(* PLC project Traffic control simulator, CODESYS CODESYS V3.5 SP14 Patch 1, author Toni Kucic *)
(* stored: creationDateTime 2019-08-10T15:27:01.2415123, version 1.0, modificationDateTime 2019-08-10T15:27:01.0436346, organization TK Automation *)

FUNCTION_BLOCK CollisionDetection
  VAR_INPUT
    xcor1 : REAL := 0;  (* X Coordinate of object 1 *)
    ycor1 : REAL := 0;  (* Y Coordinate of object 1 *)
    height1 : REAL := 0;  (* Height of object 1 *)
    width1 : REAL := 0;  (* Width of object 1 *)
    xcor2 : REAL := 0;  (* X Coordinate of object 2 *)
    ycor2 : REAL := 0;  (* Y Coordinate of object 2 *)
    height2 : REAL := 0;  (* Height of object 1 *)
    width2 : REAL := 0;  (* Width of object 1 *)
  END_VAR
  VAR_OUTPUT
    isCollision : BOOL := FALSE;
  END_VAR

            IF xcor1 < (xcor2 + width2) AND
   (xcor1 + width1) > xcor2 AND
   ycor1 < (ycor2 + height2) AND
  ( height1 + ycor1) > ycor2 THEN
   isCollision := TRUE;
ELSE
	isCollision := FALSE;
END_IF
          
END_FUNCTION_BLOCK

FUNCTION_BLOCK MoveSprite
  VAR_IN_OUT
    xCor : INT := 0;
    yCor : INT := 0;
  END_VAR
  VAR_INPUT
    xScreen : INT := 0;  (* Width of the screen *)
    yScreen : INT := 0;  (* Height of the screen *)
    SpriteWidth : INT := 0;  (* Width of the sprite *)
    SpriteHeight : INT := 0;  (* Height of the sprite *)
    ySpeed : INT := 0;  (* Control up or down movement with +- *)
    xSpeed : INT := 0;  (* Control left or right movement with +- *)
  END_VAR

            (* Reseting the position if sprite goes off screen *)
(* If moving left to right *)
IF xCor >= xScreen  AND xSpeed > 0 THEN
	xCor := -SpriteWidth;
(* If moving right to left *)
ELSIF xCor <= -SpriteWidth AND xSpeed < 0 THEN
	xCor := xScreen;	
END_IF
(* If moving from up, down *)
IF yCor >= yScreen AND ySpeed > 0 THEN
	yCor := -SpriteHeight;
(* If moving from down, up *)
ELSIF yCor < -SpriteHeight AND ySpeed < 0 THEN
	yCor := yScreen;	
END_IF

(* Actual moving of the coordinates *)
xCor := xCor + xSpeed;
yCor := yCor + ySpeed;

          
END_FUNCTION_BLOCK

PROGRAM xc03_TrafficControl
  VAR
    vSequenceA : DINT := 1;
    TimerA : TOF;
    vSequenceB : DINT := 0;
    TimerB : TOF;
    Start : BOOL;
    StartOld : BOOL;
    vSequence : DINT := 0;
    TactTimer : TON;
    vPeriodTime : TIME := TIME#1m25s0ms;
    vElapsedTime : TIME;
  END_VAR

                    
TactTimer(IN:=TRUE, PT:=vPeriodTime, ET => vElapsedTime);
IF TactTimer.Q THEN
	TactTimer(IN:=FALSE);
END_IF
(* Direction Up, Down traffic light *)
xgv03.TLight3Red := vElapsedTime <= T#5S OR vElapsedTime >= T#37S AND vElapsedTime <= T#85S;
xgv03.TLight3Yellow := vElapsedTime > T#3S AND vElapsedTime <= T#5S OR vElapsedTime >= T#35S AND vElapsedTime <= T#37S;
xgv03.TLight3Green := vElapsedTime >= T#5S AND vElapsedTime <= T#35S;

(* Mirror the other side of the Up, Down direction *)
xgv03.TLight4Red := xgv03.TLight3Red;
xgv03.TLight4Yellow := xgv03.TLight3Yellow;
xgv03.TLight4Green := xgv03.TLight3Green;

(* Direction Left, Right traffic light *)
xgv03.TLight2Red := vElapsedTime >= T#0S AND vElapsedTime <= T#39S OR vElapsedTime >= T#71S AND vElapsedTime <= T#85S;
xgv03.TLight2Yellow := vElapsedTime > T#37S AND vElapsedTime <= T#39S OR vElapsedTime >= T#69S AND vElapsedTime <= T#71S;
xgv03.TLight2Green := vElapsedTime >= T#39S AND vElapsedTime <= T#69S;

(* Mirror the other side of the Left, Right direction *)
xgv03.TLight1Red := xgv03.TLight2Red;
xgv03.TLight1Yellow := xgv03.TLight2Yellow;
xgv03.TLight1Green := xgv03.TLight2Green;
(*CASE vSequence OF
	0:
	(* Starting sequence, direction Up, Down *)
	TimerA
	Task03GVL.TLight1Red := TRUE;
	
END_CASE
CASE vSequenceA OF
	0: TimerA(IN:=FALSE,PT:=T#20S);
	Task03GVL.TLight1Yellow:= FALSE;
	Task03GVL.TLight1Red:= FALSE;
	Task03GVL.TLight1Green:= TimerA.Q;
	Task03GVL.TLight2Green := Task03GVL.TLight1Green;
	IF NOT TimerA.Q THEN
		TimerA(IN:=TRUE);
		vSequenceA:=1;
	END_IF
	1: TimerA(IN:=FALSE,PT:=T#4S);
	Task03GVL.TLight1Red:= FALSE;
	Task03GVL.TLight1Green:= FALSE;
	Task03GVL.TLight1Yellow:= TimerA.Q;
	Task03GVL.TLight2Yellow := Task03GVL.TLight1Yellow;
	IF NOT TimerA.Q THEN
		TimerA(IN:=TRUE);
		vSequenceA:=2;
	END_IF
		2: TimerA(IN:=FALSE,PT:=T#30S);
	Task03GVL.TLight1Green:= FALSE;
	Task03GVL.TLight1Yellow:= FALSE;
	Task03GVL.TLight1Red:= TimerA.Q;
	Task03GVL.TLight2Red := Task03GVL.TLight1Red;
	IF NOT TimerA.Q THEN
		TimerA(IN:=TRUE);
		vSequenceA:=3;
	END_IF
		3: TimerA(IN:=FALSE,PT:=T#4S);
	Task03GVL.TLight1Green:= FALSE;
	Task03GVL.TLight1Red:= TimerA.Q;
	Task03GVL.TLight1Yellow:= TimerA.Q;
	Task03GVL.TLight2Red := Task03GVL.TLight1Red;
	Task03GVL.TLight2Yellow := Task03GVL.TLight1Yellow;
	IF NOT TimerA.Q THEN
		TimerA(IN:=TRUE);
		vSequenceA:=0;
		IF vSequenceB=6 THEN
		vSequenceB:=3;	
		END_IF
		
	END_IF
END_CASE

CASE vSequenceB OF
	0: TimerB(IN:=FALSE,PT:=T#4S);
	Task03GVL.TLight3Green:= FALSE;
	Task03GVL.TLight3Red:= TimerB.Q;
	Task03GVL.TLight3Yellow:= TimerB.Q;
	Task03GVL.TLight4Red := Task03GVL.TLight3Red;
	Task03GVL.TLight4Yellow := Task03GVL.TLight3Yellow;
	IF NOT TimerB.Q THEN
		TimerB(IN:=TRUE);
		vSequenceB:=1;
	END_IF
	
	1: TimerB(IN:=FALSE,PT:=T#20S);
	Task03GVL.TLight3Yellow:= FALSE;
	Task03GVL.TLight3Red:= FALSE;
	Task03GVL.TLight3Green:= TimerB.Q;
	Task03GVL.TLight4Green := Task03GVL.TLight3Green;
	IF NOT TimerB.Q THEN
		TimerB(IN:=TRUE);
		vSequenceB:=2;
	END_IF
	
	2: TimerB(IN:=FALSE,PT:=T#4S);
	Task03GVL.TLight3Red:= FALSE;
	Task03GVL.TLight3Green:= FALSE;
	Task03GVL.TLight3Yellow:= TimerB.Q;
	Task03GVL.TLight4Yellow := Task03GVL.TLight3Yellow;
	IF NOT TimerB.Q THEN
		TimerB(IN:=TRUE);
		vSequenceB:=3;
	END_IF
	
		3: TimerB(IN:=FALSE,PT:=T#30S);
	Task03GVL.TLight3Green:= FALSE;
	Task03GVL.TLight3Yellow:= FALSE;
	Task03GVL.TLight3Red:= TimerB.Q;
	Task03GVL.TLight4Red := Task03GVL.TLight3Red;
	IF NOT TimerB.Q THEN
		TimerB(IN:=TRUE);
		vSequenceB:=0;
	END_IF
		
END_CASE
END_IF;*)
                  
END_PROGRAM

PROGRAM xsim03
  VAR
    Car1X : INT := 925;  (* Red car *)
    Car1Y : INT := 740;
    Car1Width : INT := 100;
    Car1Height : INT := 230;
    Car2X : INT := 420;  (* Blue car *)
    Car2Y : INT := 511;
    Car2Width : INT := 230;
    Car2Height : INT := 100;
    Car3X : INT := 1160;  (* Green car *)
    Car3Y : INT := 366;
    Car3Width : INT := 230;
    Car3Height : INT := 100;
    Car4X : INT := 775;  (* Yellow car *)
    Car4Y : INT := 0;
    Car4Width : INT := 100;
    Car4Height : INT := 230;
    Speed : INT := 1;
    vCarCrash : BOOL;
    vReset : BOOL;
    xExplosion : INT;
    yExplosion : INT;
    Car3Car4Coll : CollisionDetection;
    Car3Car1Coll : CollisionDetection;
    Car2Car1Coll : CollisionDetection;
    Car2Car4Coll : CollisionDetection;
    MoveCar1 : MoveSprite;
    MoveCar2 : MoveSprite;
    MoveCar3 : MoveSprite;
    MoveCar4 : MoveSprite;
  END_VAR

                    (* Collision detection *)
(* Car3 and Car 4 *)
Car3Car4Coll(
	xcor1:= Car3X, 
	ycor1:= Car3Y, 
	height1:= Car3Height, 
	width1:= Car3Width, 
	xcor2:= Car4X, 
	ycor2:= Car4Y, 
	height2:= Car4Height, 
	width2:= Car4Width);
(* Car3 and Car 1 *)
Car3Car1Coll(
	xcor1:= Car3X, 
	ycor1:= Car3Y, 
	height1:= Car3Height, 
	width1:= Car3Width, 
	xcor2:= Car1X, 
	ycor2:= Car1Y, 
	height2:= Car1Height, 
	width2:= Car1Width);
(* Car2 and Car 4 *)
Car2Car4Coll(
	xcor1:= Car2X, 
	ycor1:= Car2Y, 
	height1:= Car2Height, 
	width1:= Car2Width, 
	xcor2:= Car4X, 
	ycor2:= Car4Y, 
	height2:= Car4Height, 
	width2:= Car4Width);
(* Car2 and Car 1 *)
Car2Car1Coll(
	xcor1:= Car2X, 
	ycor1:= Car2Y, 
	height1:= Car2Height, 
	width1:= Car2Width, 
	xcor2:= Car1X, 
	ycor2:= Car1Y, 
	height2:= Car1Height, 
	width2:= Car1Width);

IF Car3Car4Coll.isCollision OR Car3Car1Coll.isCollision OR Car2Car4Coll.isCollision OR Car2Car1Coll.isCollision THEN
	vCarCrash := TRUE;
ELSE
	vCarCrash := FALSE;	
END_IF

(* Explosion graphic *)
IF Car3Car4Coll.isCollision THEN
	xExplosion := Car3X;
	yExplosion := Car3Y;
ELSIF Car3Car1Coll.isCollision THEN
	xExplosion := Car3X;
	yExplosion := Car3Y;
ELSIF Car2Car4Coll.isCollision THEN
	xExplosion := Car2X + Car2Width;
	yExplosion := Car2Y;
ELSIF Car2Car1Coll.isCollision THEN
	xExplosion := Car2X + Car2Width;
	yExplosion := Car2Y;
ELSE
	xExplosion := 2000;
	yExplosion := 2000;
END_IF

(* Car movements *)
IF  vCarCrash THEN
	//wait
	IF vReset THEN
		(* Reset to start position *)
		Car1X:= 925;
		Car1Y:= 740;
		Car2X:= 420;
		Car2Y:= 511;
		Car3X:= 1160;
		Car3Y:= 366;
		Car4X:= 775;
		Car4Y:= 0;
	END_IF
ELSE
	(* Define what cars do depending on lights *)
	(* car moves if its green for him or he is past the traffic ligght but stops at the traffic light if its red, or yellow.*)
	IF xgv03.TLight4Green OR Car1Y - 740 < 0 OR Car1Y - 740 > Speed THEN
		MoveCar1(
		xCor:= Car1X, 
		yCor:= Car1Y, 
		xScreen:= 1830, 
		yScreen:= 930,
		SpriteWidth:= Car1Width, 
		SpriteHeight:= Car1Height, 
		ySpeed:= -Speed, 
		xSpeed:= 0 );
	END_IF;
	IF xgv03.TLight2Green OR Car2X - 420 < 0 OR Car2X - 420 > Speed THEN
		MoveCar2(
		xCor:= Car2X, 
		yCor:= Car2Y, 
		xScreen:= 1830, 
		yScreen:= 930,
		SpriteWidth:= Car2Width, 
		SpriteHeight:= Car2Height,  
		ySpeed:= 0, 
		xSpeed:= Speed );
	END_IF;
	IF xgv03.TLight1Green OR Car3X - 1160 < 0 OR Car3X - 1160 > Speed THEN
		MoveCar3(
		xCor:= Car3X, 
		yCor:= Car3Y, 
		xScreen:= 1830, 
		yScreen:= 930,
		SpriteWidth:= Car3Width, 
		SpriteHeight:= Car3Height,  
		ySpeed:= 0, 
		xSpeed:= -Speed );
	END_IF;
	IF xgv03.TLight3Green OR Car4Y - 0 < 0 OR Car4Y - 0 > Speed THEN
		MoveCar4(
		xCor:= Car4X, 
		yCor:= Car4Y, 
		xScreen:= 1830, 
		yScreen:= 930,
		SpriteWidth:= Car4Width, 
		SpriteHeight:= Car4Height,  
		ySpeed:= Speed, 
		xSpeed:= 0 );
	END_IF;
END_IF


                  
END_PROGRAM

CONFIGURATION SoftPLC
  RESOURCE Application ON PLC
    {attribute 'qualified_only'}
    VAR_GLOBAL  (* xgv03 *)
      cfgPeriodTime : TIME := TIME#1m24s0ms;  (* Configuration *)
      cfgStartDirection : DINT := 0;
      TLight1Red : BOOL;  (* DIGITAL OUTPUT Activate red light traffic light 1 *)
      TLight1Yellow : BOOL;  (* DIGITAL OUTPUT Activate yellow light traffic light 1 *)
      TLight1Green : BOOL;  (* DIGITAL OUTPUT Activate green light traffic light 1 *)
      TLight2Red : BOOL;  (* DIGITAL OUTPUT Activate red light traffic light 2 *)
      TLight2Yellow : BOOL;  (* DIGITAL OUTPUT Activate yellow light traffic light 2 *)
      TLight2Green : BOOL;  (* DIGITAL OUTPUT Activate green light traffic light 2 *)
      TLight3Red : BOOL;  (* DIGITAL OUTPUT Activate red light traffic light 3 *)
      TLight3Yellow : BOOL;  (* DIGITAL OUTPUT Activate yellow light traffic light 3 *)
      TLight3Green : BOOL;  (* DIGITAL OUTPUT Activate green light traffic light 3 *)
      TLight4Red : BOOL;  (* DIGITAL OUTPUT Activate red light traffic light 4 *)
      TLight4Yellow : BOOL;  (* DIGITAL OUTPUT Activate yellow light traffic light 4 *)
      TLight4Green : BOOL;  (* DIGITAL OUTPUT Activate green light traffic light 4 *)
    END_VAR
    TASK VISU_TASK(INTERVAL := T#50ms, PRIORITY := 31);
    TASK xsim03(INTERVAL := T#5ms, PRIORITY := 1);
    TASK xc03_Task(INTERVAL := T#50ms, PRIORITY := 1);
    PROGRAM VisuElems.Visu_Prg WITH VISU_TASK : VisuElems.Visu_Prg;
    PROGRAM xsim03 WITH xsim03 : xsim03;
    PROGRAM xc03_TrafficControl WITH xc03_Task : xc03_TrafficControl;
  END_RESOURCE
END_CONFIGURATION
